// TIA Portal V16 export
// export: Created 2024-12-03T15:41:45.2847935Z, ExportSetting WithReadOnly, DisplayName Totally Integrated Automation Portal, DisplayVersion V16 Update 6, DisplayName TIA Portal Version Control Interface, DisplayVersion V16 Update 2, DisplayName TIA Portal Openness, DisplayVersion V16 Update 6, DisplayName TIA Portal Teamcenter Gateway, DisplayVersion V16, DisplayName SINAMICS Startdrive Advanced, DisplayVersion V16 Update 5, DisplayName SINAMICS Startdrive G130, G150, S120, S150, SINAMICS MV, S210, DisplayVersion V16 Update 5, DisplayName SINAMICS Startdrive G110M, G120, G120C, G120D, G120P, G115D, DisplayVersion V16 Update 5, DisplayName STEP 7 Professional, DisplayVersion V16 Update 6, DisplayName STEP 7 Safety, DisplayVersion V16, DisplayName WinCC Advanced / Unified PC, DisplayVersion V16 Update 6
TYPE "COGNEX_DATAMAN_OUT_UDT"
// stored: CreationDate 2022-02-10T08:20:21.8932261Z, InterfaceModifiedDate 2020-06-23T05:39:39.7523029Z, IsConsistent true, LibraryConformanceStatus The object is library-conformant., ModifiedDate 2020-06-23T22:30:53.6264385Z
   STRUCT
      TriggerContr_TriggerEnable : Bool;   // 0 = Trigger via PhotoEye1 = Trigger via Fieldbus
      TriggerContr_Trigger : Bool;   // 0 = Trigger OFF1 = Trigger ON* only when Trigger Enable == 1
      TriggerContr_Spare_2 : Bool;
      TriggerContr_Spare_3 : Bool;
      TriggerContr_ForceRunMode : Bool;   // 0 = Allow to open Setup Tool Connection1 = Block Setup Tool Connection and stay in RunMode
      TriggerContr_TriggerSetting : Bool;   // 0 = Individual Trigger per reader1 = Trigger = triggers both readers* Only for Trigger 2
      TriggerContr_TriggerPin : Bool;   // 0 = Pin 4 IN11 = Pin 2 IN2
      TriggerContr_TriggerEdge : Bool;   // 0 = Rising edge1 = Falling edge
      ResultContr_ResultAck : Bool;   // Bit is used to acknowledge that the PLC hassuccessfully read the last result data. When set to truethe ‘Result Available’ bit will be cleared.
      ResultContr_spare_1 : Bool;
      ResultContr_spare_4 : Bool;
      ResultContr_spare_6 : Bool;
      ResultContr_spare_7 : Bool;
      ResultContr_spare_8 : Bool;
      ResultContr_spare_9 : Bool;
      ResultContr_spare_10 : Bool;
      SoftEventContr_TrainCode : Bool;
      SoftEventContr_TrainMatchString : Bool;
      SoftEventContr_Focus : Bool;
      SoftEventContr_TrainBirghtness : Bool;
      SoftEventContr_Untrain : Bool;
      SoftEventContr_SetInputString : Bool;
      SoftEventContr_ExecuteDMCC : Bool;
      SoftEventContr_SetMatchString : Bool;
      UserDataOption : Int;   // Only used by “Set Match String” soft event. Specifieswhich code target to assign the string (16-bit integer)
      spare_5 : Byte;
      DataBlock_DataBlockSize_0 : Bool;
      DataBlock_DataBlockSize_1 : Bool;
      DataBlock_DataBlockSize_2 : Bool;
      DataBlock_DataBlockSize_3 : Bool;
      DataBlock_spare_4 : Bool;
      DataBlock_spare_5 : Bool;
      DataBlock_spare_6 : Bool;
      DataBlock_Reader2Disabled : Bool;   // 0 = Reader 2 Enabled (default)1 = Reader 2 Disabled
      UserData : Array[0..15] of Byte;
   END_STRUCT;
END_TYPE
